(*

## Short summary
This interface provides assert statements for floatings (``REAL`` and ``LREAL``)
For 32 bit floats (``REAL``) use `IFloatAssertions.single`
For 64 bit floats (``LREAL``) use `IFloatAssertions.double`

.. <legal notes>

legal notes
=================
| SPDX-FileCopyrightText: © 2022 ekvip automation GmbH <info@ekvip.de>
| SPDX-License-Identifier: Apache-2.0
| For details check: Apache-2.0_

.. _Apache-2.0: https://www.apache.org/licenses/LICENSE-2.0

.. </legal notes>



*)

INTERFACE IFloatAssertions EXTENDS __SYSTEM.IQueryInterface

(*

## Short summary
Returns the interface `ILrealAssertions` with assert statements for 64 bit floatings (``LREAL``)

.. <legal notes>

legal notes
=================
| SPDX-FileCopyrightText: © 2022 ekvip automation GmbH <info@ekvip.de>
| SPDX-License-Identifier: Apache-2.0
| For details check: Apache-2.0_

.. _Apache-2.0: https://www.apache.org/licenses/LICENSE-2.0

.. </legal notes>

*)

PROPERTY double :ILrealAssertions
GET
END_GET
END_PROPERTY

(*

## Short summary
Returns the interface `IRealAssertions` with assert statements for 32 bit floatings (``REAL``)

.. <legal notes>

legal notes
=================
| SPDX-FileCopyrightText: © 2022 ekvip automation GmbH <info@ekvip.de>
| SPDX-License-Identifier: Apache-2.0
| For details check: Apache-2.0_

.. _Apache-2.0: https://www.apache.org/licenses/LICENSE-2.0

.. </legal notes>

*)

PROPERTY single :IRealAssertions
GET
END_GET
END_PROPERTY

END_INTERFACE

(* stored: Version 1.1.0.1, ProductVersion 3.1.4026.11
   Itf IFloatAssertions: Id {2fd29953-0530-4853-9ac7-509f41ef4bc7}
   Property double: Id {53c39a10-3241-4905-a595-6ec1c7255a30}
   Get Get: Id {0862a99e-0941-4c9e-8a3f-92d7e6eb36c3}
   Property single: Id {4b05eb65-ef33-4f48-ba0c-65484232ed25}
   Get Get: Id {da44898d-69dc-4a13-b44f-79d82d1a4497} *)
